// TIA Portal V16 export
// export: Created 2022-06-23T08:01:19.1046953Z, ExportSetting WithDefaults, DisplayName Totally Integrated Automation Portal, DisplayVersion V16, DisplayName TIA Portal Version Control Interface, DisplayVersion V16, DisplayName TIA Portal Openness, DisplayVersion V16, DisplayName STEP 7 Professional, DisplayVersion V16, DisplayName STEP 7 Safety, DisplayVersion V16, DisplayName WinCC Advanced, DisplayVersion V16
ORGANIZATION_BLOCK "Main"   // OB1, LAD, ProgramCycle
TITLE = "Main Program Sweep (Cycle)"
{ S7_Optimized_Access := 'TRUE' }
VERSION : 0.1
// stored: AutoNumber true, IsIECCheckEnabled false, SetENOAutomatically false
   VAR_INPUT
      Initial_Call : Bool;   // Initial call of this OB
      Remanence : Bool;   // =True, if remanent data are available
   END_VAR
BEGIN

REGION Network 1
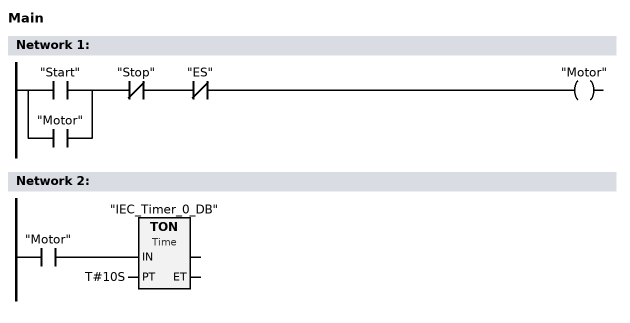
   RUNG wire#powerrail
      Contact( "Start" )
      wire#w1
      I_Contact( "Stop" )
      I_Contact( "ES" )
      Coil( "Motor" )
   END_RUNG
   RUNG wire#powerrail
      Contact( "Motor" )
   END_RUNG wire#w1
   // the same network as SCL:
   "Motor" := ("Start" OR "Motor") AND NOT "Stop" AND NOT "ES";
END_REGION

REGION Network 2
   RUNG wire#powerrail
      Contact( "Motor" )
      { S7_Templates := "time_type := Time" } "IEC_Timer_0_DB".TON(pt := T#10S, et =>)
   END_RUNG
   // the same network as SCL:
   "IEC_Timer_0_DB".TON(IN := "Motor", PT := T#10S);
END_REGION
END_ORGANIZATION_BLOCK
